// TwinCAT 3 PLC project TemperatureProject
// ProgramVersion: 3.1.4020.4
// libraries:
//   Tc2_Standard, * (Beckhoff Automation GmbH)
//   Tc2_System, * (Beckhoff Automation GmbH)
//   Tc3_Module, * (Beckhoff Automation GmbH)
// project tree:
//   / PlcTask.TcTTO
//   POUs/ MAIN.TcPOU
// real-time tasks:
//   TASK PlcTask: cycle T#10ms, priority 20, ADS port 350
// I/O:
//   DEVICE Device 1 (EtherCAT), AmsNetId 5.37.100.170.2.1
//     Term 1 (EK1200) [EK1200-5000 EtherCAT Power supply (2A E-Bus)]
//       Term 2 (EL3201) [EL3201 1Ch. Ana. Input PT100 (RTD)]
//       Term 3 (EL3064) [EL3064 4Ch. Ana. Input 0-10V]
//       Term 4 (EL9011) [EL9011 End Terminal]
// variable links:
//   TemperatureProject/TemperatureProject Instance <-> Device 1 (EtherCAT)/Term 1 (EK1200)/Term 2 (EL3201)
//     PlcTask Inputs/MAIN.aiTemperature <-> RTD/Value

CONFIGURATION TemperatureProject
    RESOURCE PLC ON TwinCAT3
        TASK PlcTask(INTERVAL := T#10ms, PRIORITY := 20);
        PROGRAM MAIN WITH PlcTask : MAIN;
    END_RESOURCE
END_CONFIGURATION

// ---- POUs/MAIN.TcPOU
PROGRAM MAIN
VAR
	aiTemperature AT %I* : INT; // Declaration of Temperature
	{attribute 'OPC.UA.DA' := '1'}
	nAlive : UDINT;
	{attribute 'OPC.UA.DA' := '1'}
	iScaledTemp : REAL;
END_VAR

iScaledTemp := INT_TO_REAL(aiTemperature) / 10;
nAlive := nAlive + 1;
IF nAlive = 10000 THEN
	nAlive := 0;
END_IF

END_PROGRAM
